// TIA Portal V16 export
// export: Created 2024-09-05T17:40:13.6595863Z, ExportSetting WithDefaults, DisplayName Totally Integrated Automation Portal, DisplayVersion V16 Update 6, DisplayName TIA Portal Version Control Interface, DisplayVersion V16 Update 2, DisplayName TIA Portal Openness, DisplayVersion V16 Update 6, DisplayName STEP 7 Professional, DisplayVersion V16 Update 6, DisplayName STEP 7 Safety, DisplayVersion V16, DisplayName WinCC Advanced, DisplayVersion V16 Update 6
TYPE "UDT_ShiftStatus"
// stored: IsFailsafeCompliant false
   STRUCT
      ShiftNumber : UInt;   // Actual shift number
      ShiftActive : Bool;   // Some shift is active
      Shift1Started : Bool;   // Shift 1 started
      Shift2Started : Bool;   // Shift 2 started
      Shift3Started : Bool;   // Shift 3 started
   END_STRUCT;
END_TYPE
